INTERFACE I_Pushbutton

PROPERTY IsPressed : BOOL
GET
END_GET
END_PROPERTY

PROPERTY IsReleased : BOOL
GET
END_GET
END_PROPERTY

END_INTERFACE

(* stored: Version 1.1.0.1, ProductVersion 3.1.4024.9
   Itf I_Pushbutton: Id {479e7ec4-eb1d-439c-8457-e6cccfb90e2e}
   Property IsPressed: Id {9cb6a6f2-4064-4dde-9d16-3e783a226f76}
   Get Get: Id {222a199d-4aca-4446-b29a-13d8358b51a6}
   Property IsReleased: Id {c34fc39f-16c9-489e-9258-e12656084724}
   Get Get: Id {fa16fd21-66e4-466f-bab2-a28b46ef9dbd} *)
